Fanuc TP program (LS listing): hmioapp6.ls

/PROG  HMIOAPP6	  Macro
/ATTR
OWNER		= RIVIAN;
COMMENT		= "Hm I-O App6 V1.0";
PROG_SIZE	= 442;
CREATE		= DATE 21-07-09  TIME 07:31:40;
MODIFIED	= DATE 21-07-09  TIME 07:31:40;
FILE_NAME	= HMIOAPP6;
VERSION		= 10;
LINE_COUNT	= 9;
MEMORY_SIZE	= 778;
PROTECT		= READ_WRITE;
TCD:  STACK_SIZE	= 0,
      TASK_PRIORITY	= 50,
      TIME_SLICE	= 0,
      BUSY_LAMP_OFF	= 0,
      ABORT_REQUEST	= 0,
      PAUSE_REQUEST	= 0;
DEFAULT_GROUP	= *,*,*,*,*;
CONTROL_CODE	= 00001000 00000000;
/APPL
/MN
   1:  !******************************** ;
   2:  ! RIVIAN AUTOMOTIVE ;
   3:  !******************************** ;
   4:  ! Set At Home I-O At Home ;
   5:  ! APP6 - ;
   6:  ! Version 1.0 ;
   7:  !******************************** ;
   8:   ;
   9:   ;
/POS
/END
